Fanuc KAREL source: kt00474.KL

-- PROVISIONAL review KL for V940-1; original PC SHA256 44f127a52a87d8757455bf46d20b40f1060c3d4958b7f46d66e0fe45ed3ddfc7
-- Incomplete behavior may be omitted. Consult companion uncertainty JSON. Do not deploy.
PROGRAM KT00474
%NOLOCKGROUP
-- UNRESOLVED_DECL P1 type=000101
-- UNRESOLVED_DECL P2 type=000101
-- UNRESOLVED_DECL OUT type=000101
BEGIN
  -- V9_ZERO_TABLE_METADATA_HINT layout=0001; no indexed target words; source/name/runtime held
  -- UNRESOLVED_PC offsets 5-29; opcodes 49,49,60,4A
  -- UNRESOLVED_PC offsets 34-38; opcodes 7F
END KT00474
